Fanuc KAREL source: kb00192.KL

-- PROVISIONAL review KL for V940-1; original PC SHA256 12ce547d80e639a3aa38940e126d32ccba1104cb8ce9abd7007f28c5186773cf
-- Incomplete behavior may be omitted. Consult companion uncertainty JSON. Do not deploy.
PROGRAM KB00192
%NOLOCKGROUP
VAR
  P1 : REAL
  RESULT : INTEGER
BEGIN
  -- V9_ZERO_TABLE_METADATA_HINT layout=0001; no indexed target words; source/name/runtime held
  -- UNRESOLVED_PC offsets 5-16; opcodes 2E,23
  -- UNRESOLVED_PC offsets 21-36; opcodes 27,22,76,23
  -- UNRESOLVED_PC offsets 41-45; opcodes 7F
END KB00192
